// TIA Portal V18 export
VAR_GLOBAL   // PLC tag table "Solenoid"
   Solenoid_01 AT %Q4.4 : Bool;
   Solenoid_02 AT %Q4.5 : Bool;
   Solenoid_03 AT %Q4.6 : Bool;
   Solenoid_04 AT %Q4.7 : Bool;
   Solenoid_05 AT %Q5.0 : Bool;
   Solenoid_06 AT %Q5.1 : Bool;
   Solenoid_07 AT %Q5.2 : Bool;
   Solenoid_08 AT %Q5.3 : Bool;
   Solenoid_09 AT %Q5.4 : Bool;
   Solenoid_10 AT %Q5.5 : Bool;
   Solenoid_11 AT %Q5.6 : Bool;
   Solenoid_12 AT %Q5.7 : Bool;
   Solenoid_13 AT %Q6.0 : Bool;
   Solenoid_14 AT %Q6.1 : Bool;
   Solenoid_15 AT %Q6.2 : Bool;
   Solenoid_16 AT %Q6.3 : Bool;
   Solenoid_17 AT %Q6.4 : Bool;
   Solenoid_18 AT %Q6.5 : Bool;
END_VAR
